FUNCTION CheckDivLReal : LREAL
VAR_INPUT
	divisor:LREAL;
END_VAR

{noflow}
IF divisor = 0 THEN
	CheckDivLReal:=1;
	oaksGVL.udiCheckDivLReal := oaksGVL.udiCheckDivLReal + 1;
ELSE
	CheckDivLReal:=divisor;
END_IF;
{flow}

END_FUNCTION

(* stored: Version 1.1.0.1, ProductVersion 3.1.4022.18
   POU CheckDivLReal: Id {bd38b448-914a-4b13-931c-e6ab2c6b1db8}, SpecialFunc CheckDivReal64 *)
